PROGRAM MAIN
VAR
	output1 AT %Q* : BOOL;
END_VAR

END_PROGRAM

(* stored: Version 1.1.0.1, ProductVersion 3.1.4024.2
   POU MAIN: Id {4b706781-9c08-414f-96aa-e618946640e2}, SpecialFunc None *)
